FUNCTION_BLOCK FB_SimBarcodeScanner
VAR_INPUT
END_VAR
VAR_OUTPUT
END_VAR
VAR
	bTriggerRead				AT %I* : BOOL;
	sBarcode					AT %Q* : STRING(255);
	bPartPresent				AT %Q* : BOOL;
	
	rand						: DRAND;
	fRand						: LREAL;
	tmrWork						: TON;
	iWorkMs						: DINT;
	iState						: DINT;
	iRetryCount					: DINT;
END_VAR
VAR CONSTANT
	CHANCE_NOREAD				: LREAL := 0.05;
	CHANCE_FAIL					: LREAL := 0.01;
	NO_READ						: STRING(255) := 'NO_READ';
END_VAR

rand(Seed:=107);

CASE iState OF
	0:
		IF bTriggerRead THEN
			fRand := rand.Num;
			iWorkMs := 250 + TO_DINT(fRand * 1000);
			IF rand.Num < CHANCE_FAIL THEN
				iRetryCount := 0;
				iState := 11;
			ELSE
				iState := 10;
			END_IF
		ELSE
			sBarcode := '';
		END_IF
		
	10:
		tmrWork(IN:=TRUE, PT:=TO_TIME(iWorkMs));
		IF tmrWork.Q THEN
			tmrWork(IN:=FALSE);
			IF rand.Num > CHANCE_NOREAD THEN
				sBarcode := CONCAT('BRCD_', TO_STRING(TO_DINT(fRand * 100000)));
			ELSE
				sBarcode := NO_READ;
			END_IF
			iState := 20;
		END_IF
		
	11:
		IF bTriggerRead THEN
			tmrWork(IN:=TRUE, PT:=TO_TIME(iWorkMs));
			IF tmrWork.Q THEN
				tmrWork(IN:=FALSE);
				sBarcode := NO_READ;
				iRetryCount := iRetryCount + 1;
			END_IF
		ELSE
			IF iRetryCount >= 3 THEN
				iState := 0;
			END_IF
			sBarcode := '';
		END_IF
		
		
	20:
		iState := 0;
		
END_CASE

PROPERTY PUBLIC PartPresent : BOOL
GET
PartPresent := bPartPresent;
END_GET
SET
bPartPresent := PartPresent;
END_SET
END_PROPERTY

END_FUNCTION_BLOCK

(* stored: Version 1.1.0.1, ProductVersion 3.1.4024.12
   POU FB_SimBarcodeScanner: Id {24c3bcaa-826f-4abc-9b5e-ecb042fac50e}, SpecialFunc None
   Property PartPresent: Id {20434da3-0e36-4ba4-919f-7f980e428bad}
   Get Get: Id {c5238dec-471e-4d37-815d-46cd608efa6d}
   Set Set: Id {cb171cbc-09bb-4436-b089-139751bc78fd} *)
